PROGRAM PRG_TC
VAR
END_VAR

//Measure Thercmocouples
TC_01();
TC_02();
TC_03();
TC_04();

END_PROGRAM

(* stored: Version 1.1.0.1, ProductVersion 3.1.4024.12
   POU PRG_TC: Id {af381e65-1cb1-40ba-a67a-42436983bb1f}, SpecialFunc None *)
